Staubli VAL3: makeTraj.pgx

public program makeTraj(string& x_sItem[])
  local num i
  local num l_nDistance
  local num l_nSize
  local tool l_tTool
  local bool l_bToStop
  local mdesc l_mDesc
  local num l_nMoveId
  local bool l_bOk
  local string l_sType
  local TrajectoryItem l_tTraj
  local ActionItem l_aAction
  local point l_pPoint[2]
begin
  // take the TOOL
  call tcp:getTool(l_tTool,pt:tTraj[sTrajCycle].nIndexTool)
  // the maximum size
  call getSizeItem(true,l_nSize)
  //
  // for all of my traj cyclePoints move the robot
  //
  resize(tTraj.tSuper,1,size(pt:tTraj[sTrajCycle].tData))
  for i=0 to (l_nSize-1)
    tTraj.tSuper[i]=pt:tTraj[sTrajCycle].tData[i].tSuper
  endFor
  tTraj.sID="TRAJ "+pt:tTraj[sTrajCycle].sID
  call cycleStatus:addTraj(tTraj)
  //
  // for all of my traj cyclePoints move the robot
  //
  for i=0 to (l_nSize-1)
    //
    // get the point info
    //
    l_tTraj=pt:tTraj[sTrajCycle].tData[i].tSuper
    call getPoint(l_pPoint,true,i)
    //
    // get the distance in percentage
    call getDistance(l_tTool,l_nDistance,true,i)
    //
    // give to the traj library the percentage distance
    //
    if l_bToStop
      l_tTraj.nom_speed.blend=off
    elseIf l_tTraj.moveType!=0
      l_tTraj.nom_speed.blend=Cartesian
    endIf
    //
    // put the move in the stack
    //
    switch l_tTraj.moveType
      case 0
        // or is not in range
        l_nMoveId=movej(l_pPoint,l_tTool,l_tTraj.nom_speed)
      break
      case 1
        l_nMoveId=movel(l_pPoint,l_tTool,l_tTraj.nom_speed)
      break
      case 2
        l_nMoveId=movec(l_pPoint[1],l_pPoint,l_tTool,l_tTraj.nom_speed)
      break
    endSwitch
    //
    // set the ID
    //
    l_aAction.nDistance=l_nDistance
    l_aAction.nPointId=i
    l_aAction.nMoveId=l_nMoveId
    l_aAction.sIdTraj="TRAJ "+pt:tTraj[sTrajCycle].sID
    call cycleStatus:putInstr_Traj(l_aAction,l_tTraj,pt:tTraj[sTrajCycle].nIndexTool,l_nSize)
    // there is a waitEndMove
    if l_tTraj.toStop
      waitEndMove()
      delay(l_tTraj.nStop)
      // wait all the action has been done
      wait(cycleStatus:bActionRunning==false)
    endIf
  endFor
  // bye bye
end
